FUNCTION_BLOCK SPLIT_AL_INTO_AB (* this Function splits the 8 AB (BYTE) adapters from a AL (LWORD) *)
  (* Standard: 61499-2; Description: Copyright (c) 2026 Meisterschulen am Ostbahnhof SPDX-License-Identifier: EPL-2.0 *)
  (* Version 1.0, 2026-05-16, Franz Höpfinger, Meisterschulen am Ostbahnhof, initial API and implementation and/or initial documentation *)
  PACKAGE adapter::splitting;
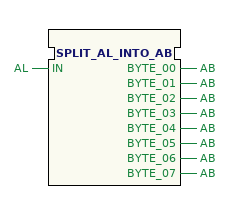
  SOCKETS
    IN : adapter::types::unidirectional::AL; (* LWORD Input *)
  END_SOCKETS
  PLUGS
    BYTE_00 : adapter::types::unidirectional::AB; (* Byte 0 *)
    BYTE_01 : adapter::types::unidirectional::AB; (* Byte 1 *)
    BYTE_02 : adapter::types::unidirectional::AB; (* Byte 2 *)
    BYTE_03 : adapter::types::unidirectional::AB; (* Byte 3 *)
    BYTE_04 : adapter::types::unidirectional::AB; (* Byte 4 *)
    BYTE_05 : adapter::types::unidirectional::AB; (* Byte 5 *)
    BYTE_06 : adapter::types::unidirectional::AB; (* Byte 6 *)
    BYTE_07 : adapter::types::unidirectional::AB; (* Byte 7 *)
  END_PLUGS
END_FUNCTION_BLOCK
